// TIA Portal V21 export
TYPE "AxixAS_DataSincro_Type_v2.0"
   STRUCT
      DataIn : "AxixAS_DataIn_Type_v2.0";
      DataOut { S7_SetPoint := 'True'} : "AxixAS_DataOut_Type_v2.0";
      ixEnableSincro { S7_SetPoint := 'True'} : Int;   // = 0 Single Axis // = 1 Master Axis // = 2 Slave Axis
      "ifDistance_Master/Slave" { S7_SetPoint := 'True'} : Real;   // Spazio cuscinetto tra Master e Slave
      ifErrorSincro { S7_SetPoint := 'True'} : Real;   // Spazio STOP istantaneo per errore
   END_STRUCT;
END_TYPE
